INTERFACE I_Crane

METHOD ControlValveOutput
VAR_INPUT
END_VAR
END_METHOD

METHOD FLOW : REAL
VAR_INPUT
END_VAR
END_METHOD

METHOD Position : ST_Position
VAR_INPUT
END_VAR
END_METHOD

METHOD Pressure : REAL
VAR_INPUT
END_VAR
END_METHOD

END_INTERFACE

(* stored: Version 1.1.0.1, ProductVersion 3.1.4024.12
   Itf I_Crane: Id {01dae7f1-e59e-41ad-b3e5-147bab081d20}
   Method ControlValveOutput: Id {7eb4ab72-8e01-4350-a744-d01a96c40922}
   Method FLOW: Id {f32959ff-f34f-4780-b7f9-aa2b2c1ef522}
   Method Position: Id {66d8546f-60ff-4d45-ab20-a28057bb29f6}
   Method Pressure: Id {d8ab2920-4eed-4dd6-a93c-596eb06fd31b} *)
